PROGRAM MAIN
VAR
	// TcUnit finds every FB_TestSuite instance by itself; it is enough to declare them here.
	fbIsNumericValueTests	: FB_IsNumericValue_Tests;
	fbEscapeInfluxTests		: FB_EscapeInfluxString_Tests;
	fbYRealTests			: FB_YREAL_Tests;
	fbTrackingTests			: FB_Tracking_Tests;
	fbPointingModelTests	: FB_PointingModel_Tests;
	fbBlinkTests			: FB_Blink_Tests;
	fbAxisTests				: FB_Axis_Tests;
	fbAstroClockSyncTests	: FB_AstroClockSync_Tests;
	fbInfluxLineProtocolTests	: FB_InfluxLineProtocol_Tests;
	fbInfluxMessageTests		: FB_InfluxMessage_Tests;
	fbCommMqttInfluxTests		: FB_Comm_MQTT_Influx_Tests;
	fbInfoConnectionTests		: FB_InfoConnection_Tests;
	fbSetpointEnableTests		: F_SetpointEnableExecute_Tests;
END_VAR

TcUnit.RUN();

END_PROGRAM

(* stored: Version 1.1.0.1, ProductVersion 3.1.4024.15
   POU MAIN: Id {cff6a572-fd5e-4250-bf6d-4eb47ba9e04d}, SpecialFunc None *)
